Universal Robots URScript: Programa_1_Iniciales_BMBL.script

def Programa_1_Iniciales_BMBL():
  sim = rpc_factory("xmlrpc", "http://172.17.0.1:40404/RPC2")
  set_tcp(p[0,0,0,0,0,0])
  set_payload(0.8, [0,0,0.04])
  movej([0, -1.570796327, 1.570796327, -1.570796327, -1.570796327, 0], a=0.6, v=0.4)
  base = get_actual_tcp_pose()
  def punto(dx, dy, dz):
    return p[base[0]+dx,base[1]+dy,base[2]+dz,base[3],base[4],base[5]]
  end
  sim.event("iniciales_iniciadas", get_actual_tcp_pose())
  popup("Letra B — inicial 1: Brayan Mateo Bravo Losada", title="Programa 1", blocking=True)
  sim.event("letra_1_B", get_actual_tcp_pose())
  movel(punto(-0.090000,-0.035000,0.03), a=0.3, v=0.08)
  movel(punto(-0.090000,-0.035000,0), a=0.3, v=0.06)
  movel(punto(-0.090000,0.035000,0), a=0.3, v=0.06)
  sim.event("trazo", get_actual_tcp_pose())
  movel(punto(-0.090000,0.035000,0.03), a=0.3, v=0.08)
  movel(punto(-0.090000,0.035000,0.03), a=0.3, v=0.08)
  movel(punto(-0.090000,0.035000,0), a=0.3, v=0.06)
  movel(punto(-0.073200,0.035000,0), a=0.3, v=0.06)
  sim.event("trazo", get_actual_tcp_pose())
  movel(punto(-0.066235,0.033668,0), a=0.3, v=0.06)
  sim.event("trazo", get_actual_tcp_pose())
  movel(punto(-0.060331,0.029874,0), a=0.3, v=0.06)
  sim.event("trazo", get_actual_tcp_pose())
  movel(punto(-0.056385,0.024197,0), a=0.3, v=0.06)
  sim.event("trazo", get_actual_tcp_pose())
  movel(punto(-0.055000,0.017500,0), a=0.3, v=0.06)
  sim.event("trazo", get_actual_tcp_pose())
  movel(punto(-0.056385,0.010803,0), a=0.3, v=0.06)
  sim.event("trazo", get_actual_tcp_pose())
  movel(punto(-0.060331,0.005126,0), a=0.3, v=0.06)
  sim.event("trazo", get_actual_tcp_pose())
  movel(punto(-0.066235,0.001332,0), a=0.3, v=0.06)
  sim.event("trazo", get_actual_tcp_pose())
  movel(punto(-0.073200,0.000000,0), a=0.3, v=0.06)
  sim.event("trazo", get_actual_tcp_pose())
  movel(punto(-0.090000,0.000000,0), a=0.3, v=0.06)
  sim.event("trazo", get_actual_tcp_pose())
  movel(punto(-0.090000,0.000000,0.03), a=0.3, v=0.08)
  movel(punto(-0.090000,0.000000,0.03), a=0.3, v=0.08)
  movel(punto(-0.090000,0.000000,0), a=0.3, v=0.06)
  movel(punto(-0.073200,0.000000,0), a=0.3, v=0.06)
  sim.event("trazo", get_actual_tcp_pose())
  movel(punto(-0.066235,-0.001332,0), a=0.3, v=0.06)
  sim.event("trazo", get_actual_tcp_pose())
  movel(punto(-0.060331,-0.005126,0), a=0.3, v=0.06)
  sim.event("trazo", get_actual_tcp_pose())
  movel(punto(-0.056385,-0.010803,0), a=0.3, v=0.06)
  sim.event("trazo", get_actual_tcp_pose())
  movel(punto(-0.055000,-0.017500,0), a=0.3, v=0.06)
  sim.event("trazo", get_actual_tcp_pose())
  movel(punto(-0.056385,-0.024197,0), a=0.3, v=0.06)
  sim.event("trazo", get_actual_tcp_pose())
  movel(punto(-0.060331,-0.029874,0), a=0.3, v=0.06)
  sim.event("trazo", get_actual_tcp_pose())
  movel(punto(-0.066235,-0.033668,0), a=0.3, v=0.06)
  sim.event("trazo", get_actual_tcp_pose())
  movel(punto(-0.073200,-0.035000,0), a=0.3, v=0.06)
  sim.event("trazo", get_actual_tcp_pose())
  movel(punto(-0.090000,-0.035000,0), a=0.3, v=0.06)
  sim.event("trazo", get_actual_tcp_pose())
  movel(punto(-0.090000,-0.035000,0.03), a=0.3, v=0.08)
  popup("Letra M — inicial 2: Brayan Mateo Bravo Losada", title="Programa 1", blocking=True)
  sim.event("letra_2_M", get_actual_tcp_pose())
  movel(punto(-0.040000,-0.035000,0.03), a=0.3, v=0.08)
  movel(punto(-0.040000,-0.035000,0), a=0.3, v=0.06)
  movel(punto(-0.040000,0.035000,0), a=0.3, v=0.06)
  sim.event("trazo", get_actual_tcp_pose())
  movel(punto(-0.022500,-0.003500,0), a=0.3, v=0.06)
  sim.event("trazo", get_actual_tcp_pose())
  movel(punto(-0.005000,0.035000,0), a=0.3, v=0.06)
  sim.event("trazo", get_actual_tcp_pose())
  movel(punto(-0.005000,-0.035000,0), a=0.3, v=0.06)
  sim.event("trazo", get_actual_tcp_pose())
  movel(punto(-0.005000,-0.035000,0.03), a=0.3, v=0.08)
  popup("Letra B — inicial 3: Brayan Mateo Bravo Losada", title="Programa 1", blocking=True)
  sim.event("letra_3_B", get_actual_tcp_pose())
  movel(punto(0.010000,-0.035000,0.03), a=0.3, v=0.08)
  movel(punto(0.010000,-0.035000,0), a=0.3, v=0.06)
  movel(punto(0.010000,0.035000,0), a=0.3, v=0.06)
  sim.event("trazo", get_actual_tcp_pose())
  movel(punto(0.010000,0.035000,0.03), a=0.3, v=0.08)
  movel(punto(0.010000,0.035000,0.03), a=0.3, v=0.08)
  movel(punto(0.010000,0.035000,0), a=0.3, v=0.06)
  movel(punto(0.026800,0.035000,0), a=0.3, v=0.06)
  sim.event("trazo", get_actual_tcp_pose())
  movel(punto(0.033765,0.033668,0), a=0.3, v=0.06)
  sim.event("trazo", get_actual_tcp_pose())
  movel(punto(0.039669,0.029874,0), a=0.3, v=0.06)
  sim.event("trazo", get_actual_tcp_pose())
  movel(punto(0.043615,0.024197,0), a=0.3, v=0.06)
  sim.event("trazo", get_actual_tcp_pose())
  movel(punto(0.045000,0.017500,0), a=0.3, v=0.06)
  sim.event("trazo", get_actual_tcp_pose())
  movel(punto(0.043615,0.010803,0), a=0.3, v=0.06)
  sim.event("trazo", get_actual_tcp_pose())
  movel(punto(0.039669,0.005126,0), a=0.3, v=0.06)
  sim.event("trazo", get_actual_tcp_pose())
  movel(punto(0.033765,0.001332,0), a=0.3, v=0.06)
  sim.event("trazo", get_actual_tcp_pose())
  movel(punto(0.026800,0.000000,0), a=0.3, v=0.06)
  sim.event("trazo", get_actual_tcp_pose())
  movel(punto(0.010000,0.000000,0), a=0.3, v=0.06)
  sim.event("trazo", get_actual_tcp_pose())
  movel(punto(0.010000,0.000000,0.03), a=0.3, v=0.08)
  movel(punto(0.010000,0.000000,0.03), a=0.3, v=0.08)
  movel(punto(0.010000,0.000000,0), a=0.3, v=0.06)
  movel(punto(0.026800,0.000000,0), a=0.3, v=0.06)
  sim.event("trazo", get_actual_tcp_pose())
  movel(punto(0.033765,-0.001332,0), a=0.3, v=0.06)
  sim.event("trazo", get_actual_tcp_pose())
  movel(punto(0.039669,-0.005126,0), a=0.3, v=0.06)
  sim.event("trazo", get_actual_tcp_pose())
  movel(punto(0.043615,-0.010803,0), a=0.3, v=0.06)
  sim.event("trazo", get_actual_tcp_pose())
  movel(punto(0.045000,-0.017500,0), a=0.3, v=0.06)
  sim.event("trazo", get_actual_tcp_pose())
  movel(punto(0.043615,-0.024197,0), a=0.3, v=0.06)
  sim.event("trazo", get_actual_tcp_pose())
  movel(punto(0.039669,-0.029874,0), a=0.3, v=0.06)
  sim.event("trazo", get_actual_tcp_pose())
  movel(punto(0.033765,-0.033668,0), a=0.3, v=0.06)
  sim.event("trazo", get_actual_tcp_pose())
  movel(punto(0.026800,-0.035000,0), a=0.3, v=0.06)
  sim.event("trazo", get_actual_tcp_pose())
  movel(punto(0.010000,-0.035000,0), a=0.3, v=0.06)
  sim.event("trazo", get_actual_tcp_pose())
  movel(punto(0.010000,-0.035000,0.03), a=0.3, v=0.08)
  popup("Letra L — inicial 4: Brayan Mateo Bravo Losada", title="Programa 1", blocking=True)
  sim.event("letra_4_L", get_actual_tcp_pose())
  movel(punto(0.060000,0.035000,0.03), a=0.3, v=0.08)
  movel(punto(0.060000,0.035000,0), a=0.3, v=0.06)
  movel(punto(0.060000,-0.035000,0), a=0.3, v=0.06)
  sim.event("trazo", get_actual_tcp_pose())
  movel(punto(0.095000,-0.035000,0), a=0.3, v=0.06)
  sim.event("trazo", get_actual_tcp_pose())
  movel(punto(0.095000,-0.035000,0.03), a=0.3, v=0.08)
  sim.event("iniciales_terminadas", get_actual_tcp_pose())
  movej([0, -1.570796327, 1.570796327, -1.570796327, -1.570796327, 0], a=0.6, v=0.4)
end
